// TIA Portal V18 export
DATA_BLOCK "Block_1_DB"   // DB1
VERSION : 0.1
// stored: AutoNumber true, InstanceOfName Block_1, InstanceOfType FB
"Block_1"
BEGIN
END_DATA_BLOCK
